// LS Electric XG5000 project: Maycatnhom_Q9
// PLC NewPLC

PROGRAM Orijine Git (task: Scan Program)

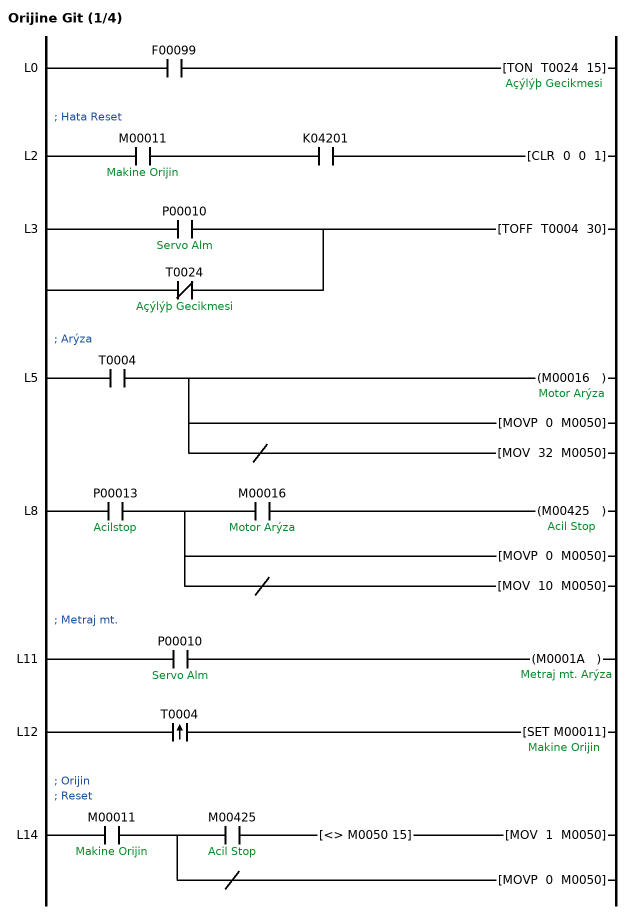
; L0
LOAD      F00099
TON       T0024 15	// Açýlýþ Gecikmesi
// Hata Reset
; L2
LOAD      M00011	// Makine Orijin
AND       K04201
CLR       0 0 1
; L3
LOAD      P00010	// Servo Alm
OR NOT    T0024	// Açýlýþ Gecikmesi
TOFF      T0004 30
; L5
LOAD      T0004
OUT       M00016	// Motor Arýza
MOVP      0 M0050
NOT
MOV       32 M0050
// output comment: Arýza
; L8
LOAD      P00013	// Acilstop
MPUSH
AND       M00016	// Motor Arýza
OUT       M00425	// Acil Stop
MPOP
MOVP      0 M0050
NOT
MOV       10 M0050
; L11
LOAD      P00010	// Servo Alm
OUT       M0001A	// Metraj mt. Arýza
// output comment: Metraj mt.
; L12
LOADP     T0004
SET       M00011	// Makine Orijin
// Orijin
; L14
LOAD      M00011	// Makine Orijin
MPUSH
AND       M00425	// Acil Stop
AND<>     M0050 15
MOV       1 M0050
MPOP
NOT
MOVP      0 M0050
// output comment: Reset

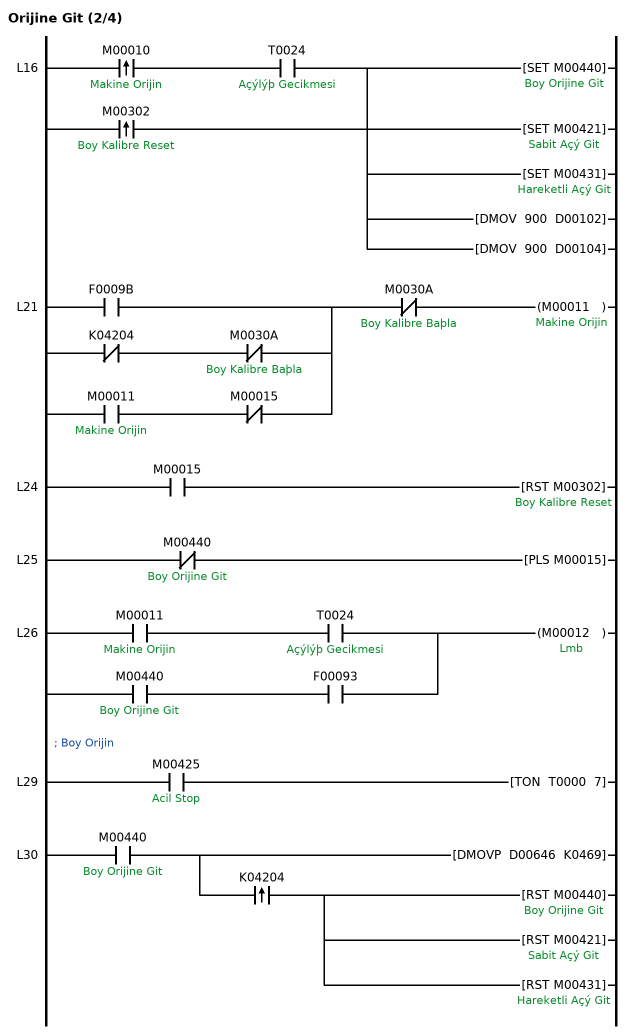
; L16
LOADP     M00010	// Makine Orijin
AND       T0024	// Açýlýþ Gecikmesi
ORP       M00302	// Boy Kalibre Reset
SET       M00440	// Boy Orijine Git
SET       M00421	// Sabit Açý Git
SET       M00431	// Hareketli Açý Git
DMOV      900 D00102
DMOV      900 D00104
; L21
LOAD      F0009B
LOAD NOT  K04204
AND NOT   M0030A	// Boy Kalibre Baþla
OR LOAD
LOAD      M00011	// Makine Orijin
AND NOT   M00015
OR LOAD
AND NOT   M0030A	// Boy Kalibre Baþla
OUT       M00011	// Makine Orijin
; L24
LOAD      M00015
RST       M00302	// Boy Kalibre Reset
; L25
LOAD NOT  M00440	// Boy Orijine Git
OUTP      M00015
; L26
LOAD      M00011	// Makine Orijin
AND       T0024	// Açýlýþ Gecikmesi
LOAD      M00440	// Boy Orijine Git
AND       F00093
OR LOAD
OUT       M00012	// Lmb
// Boy Orijin
; L29
LOAD      M00425	// Acil Stop
TON       T0000 7
; L30
LOAD      M00440	// Boy Orijine Git
DMOVP     D00646 K0469
ANDP      K04204
RST       M00440	// Boy Orijine Git
RST       M00421	// Sabit Açý Git
RST       M00431	// Hareketli Açý Git

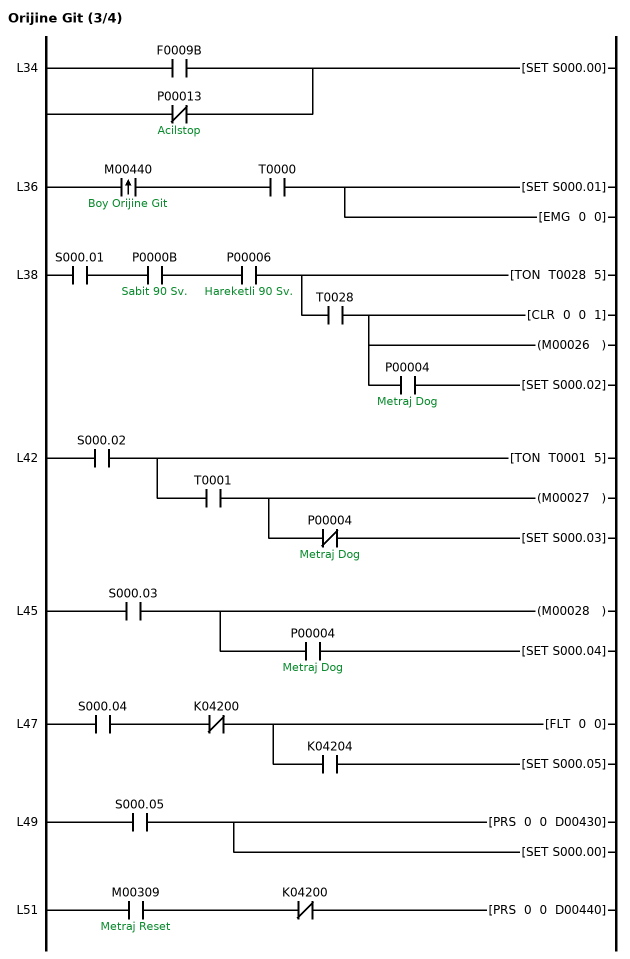
; L34
LOAD      F0009B
OR NOT    P00013	// Acilstop
SET       S000.00
; L36
LOADP     M00440	// Boy Orijine Git
AND       T0000
SET       S000.01
EMG       0 0
; L38
LOAD      S000.01
AND       P0000B	// Sabit 90 Sv.
AND       P00006	// Hareketli 90 Sv.
TON       T0028 5
AND       T0028
CLR       0 0 1
OUT       M00026
AND       P00004	// Metraj Dog
SET       S000.02
; L42
LOAD      S000.02
TON       T0001 5
AND       T0001
OUT       M00027
AND NOT   P00004	// Metraj Dog
SET       S000.03
; L45
LOAD      S000.03
OUT       M00028
AND       P00004	// Metraj Dog
SET       S000.04
; L47
LOAD      S000.04
AND NOT   K04200
FLT       0 0
AND       K04204
SET       S000.05
; L49
LOAD      S000.05
PRS       0 0 D00430
SET       S000.00
; L51
LOAD      M00309	// Metraj Reset
AND NOT   K04200
PRS       0 0 D00440

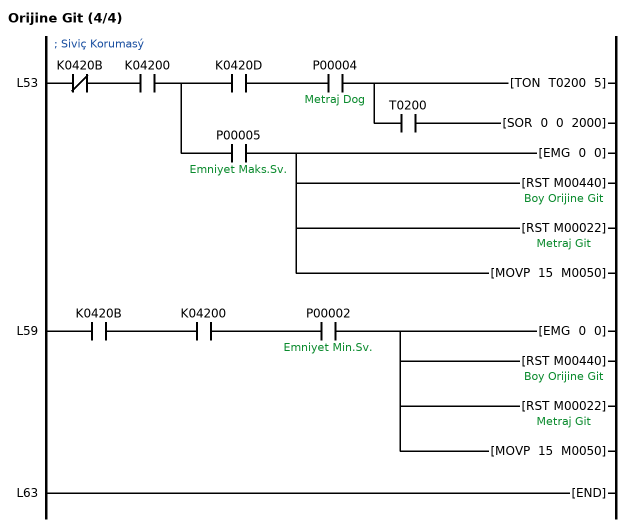
// Siviç Korumasý
; L53
LOAD NOT  K0420B
AND       K04200
MPUSH
AND       K0420D
AND       P00004	// Metraj Dog
TON       T0200 5
AND       T0200
SOR       0 0 2000
MPOP
AND       P00005	// Emniyet Maks.Sv.
EMG       0 0
RST       M00440	// Boy Orijine Git
RST       M00022	// Metraj Git
MOVP      15 M0050
; L59
LOAD      K0420B
AND       K04200
AND       P00002	// Emniyet Min.Sv.
EMG       0 0
RST       M00440	// Boy Orijine Git
RST       M00022	// Metraj Git
MOVP      15 M0050
; L63
END

PROGRAM Testere (task: Scan Program)

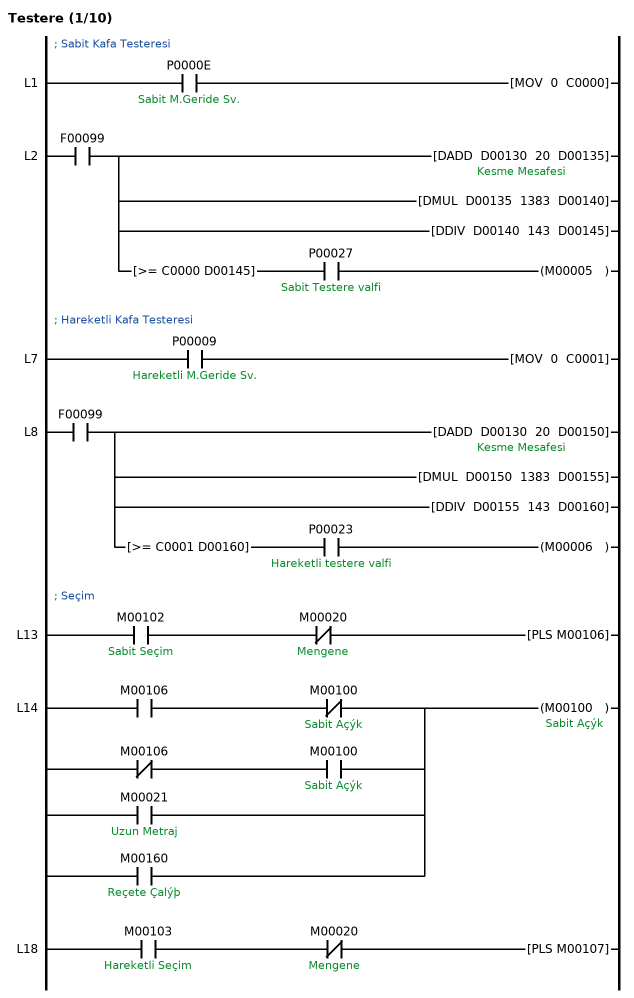
// Sabit Kafa Testeresi
; L1
LOAD      P0000E	// Sabit M.Geride Sv.
MOV       0 C0000
; L2
LOAD      F00099
DADD      D00130 20 D00135	// Kesme Mesafesi
DMUL      D00135 1383 D00140
DDIV      D00140 143 D00145
AND>=     C0000 D00145
AND       P00027	// Sabit Testere valfi
OUT       M00005
// Hareketli Kafa Testeresi
; L7
LOAD      P00009	// Hareketli M.Geride Sv.
MOV       0 C0001
; L8
LOAD      F00099
DADD      D00130 20 D00150	// Kesme Mesafesi
DMUL      D00150 1383 D00155
DDIV      D00155 143 D00160
AND>=     C0001 D00160
AND       P00023	// Hareketli testere valfi
OUT       M00006
// Seçim
; L13
LOAD      M00102	// Sabit Seçim
AND NOT   M00020	// Mengene
OUTP      M00106
; L14
LOAD      M00106
AND NOT   M00100	// Sabit Açýk
LOAD NOT  M00106
AND       M00100	// Sabit Açýk
OR LOAD
OR        M00021	// Uzun Metraj
OR        M00160	// Reçete Çalýþ
OUT       M00100	// Sabit Açýk
; L18
LOAD      M00103	// Hareketli Seçim
AND NOT   M00020	// Mengene
OUTP      M00107

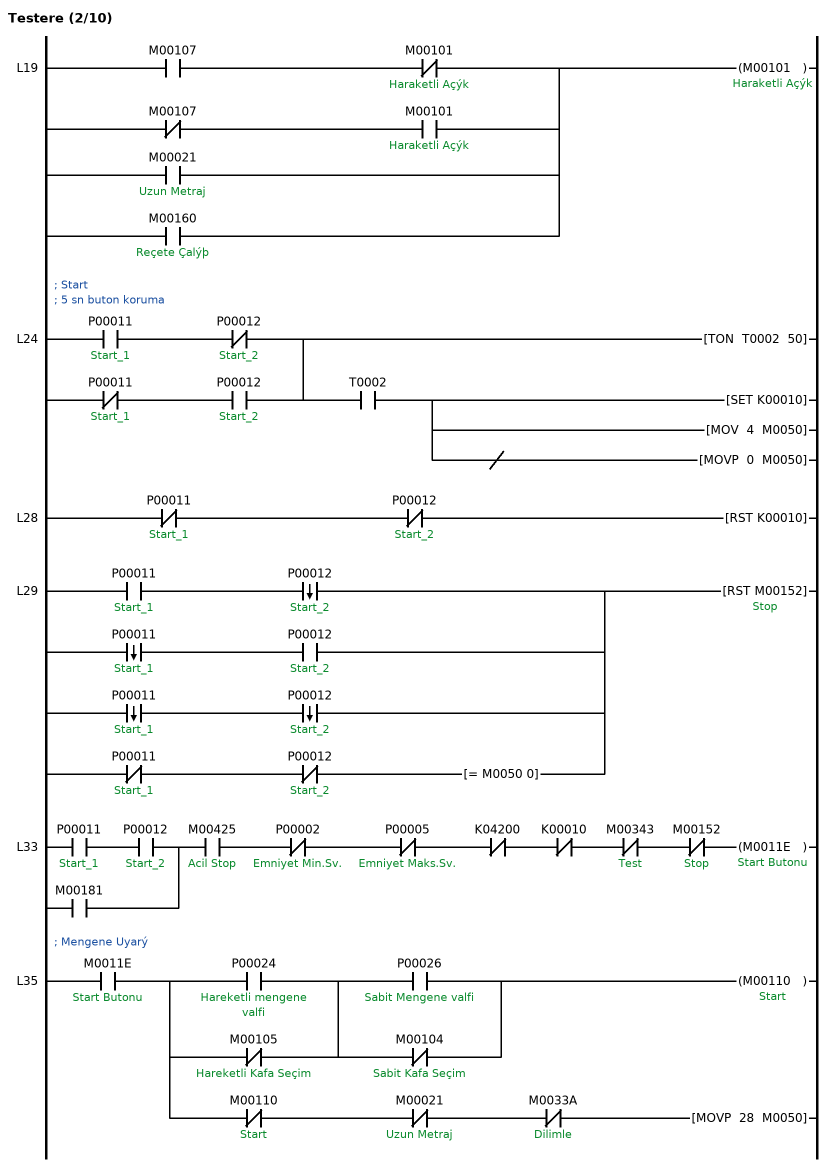
; L19
LOAD      M00107
AND NOT   M00101	// Haraketli Açýk
LOAD NOT  M00107
AND       M00101	// Haraketli Açýk
OR LOAD
OR        M00021	// Uzun Metraj
OR        M00160	// Reçete Çalýþ
OUT       M00101	// Haraketli Açýk
// Start
; L24
LOAD      P00011	// Start_1
AND NOT   P00012	// Start_2
LOAD NOT  P00011	// Start_1
AND       P00012	// Start_2
OR LOAD
TON       T0002 50
AND       T0002
SET       K00010
MOV       4 M0050
NOT
MOVP      0 M0050
// output comment: 5 sn buton koruma
; L28
LOAD NOT  P00011	// Start_1
AND NOT   P00012	// Start_2
RST       K00010
; L29
LOAD      P00011	// Start_1
ANDN      P00012	// Start_2
LOADN     P00011	// Start_1
AND       P00012	// Start_2
OR LOAD
LOADN     P00011	// Start_1
ANDN      P00012	// Start_2
OR LOAD
LOAD NOT  P00011	// Start_1
AND NOT   P00012	// Start_2
AND=      M0050 0
OR LOAD
RST       M00152	// Stop
; L33
LOAD      P00011	// Start_1
AND       P00012	// Start_2
OR        M00181
AND       M00425	// Acil Stop
AND NOT   P00002	// Emniyet Min.Sv.
AND NOT   P00005	// Emniyet Maks.Sv.
AND NOT   K04200
AND NOT   K00010
AND NOT   M00343	// Test
AND NOT   M00152	// Stop
OUT       M0011E	// Start Butonu
; L35
LOAD      M0011E	// Start Butonu
MPUSH
LOAD      P00024	// Hareketli mengene valfi
OR NOT    M00105	// Hareketli Kafa Seçim
AND LOAD
LOAD      P00026	// Sabit Mengene valfi
OR NOT    M00104	// Sabit Kafa Seçim
AND LOAD
OUT       M00110	// Start
MPOP
AND NOT   M00110	// Start
AND NOT   M00021	// Uzun Metraj
AND NOT   M0033A	// Dilimle
MOVP      28 M0050
// output comment: Mengene Uyarý

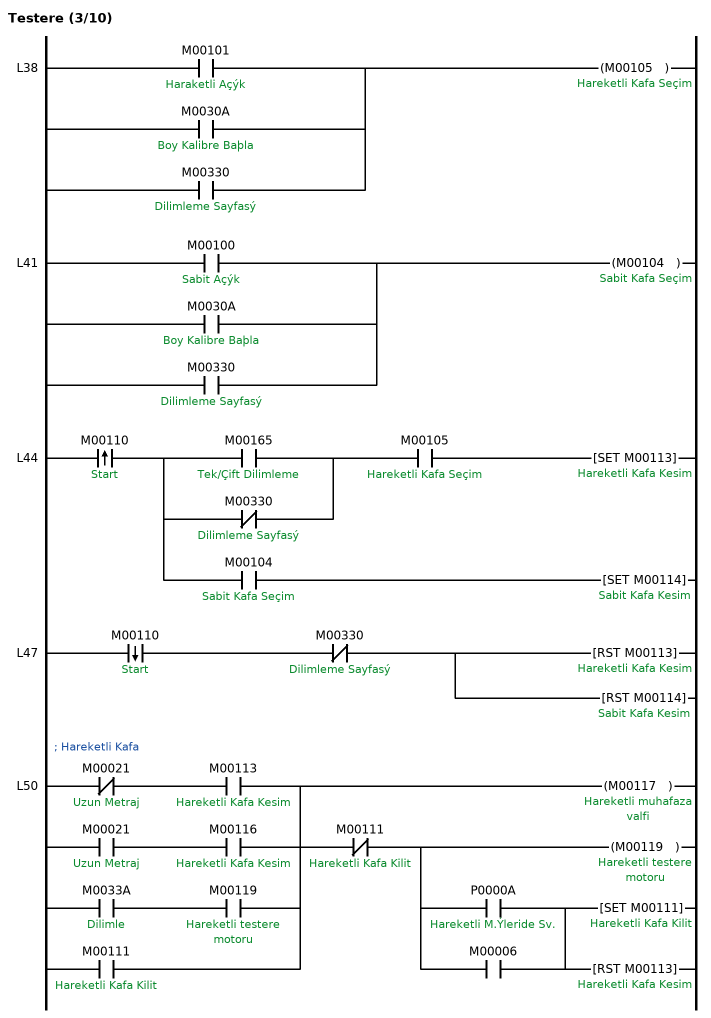
; L38
LOAD      M00101	// Haraketli Açýk
OR        M0030A	// Boy Kalibre Baþla
OR        M00330	// Dilimleme Sayfasý
OUT       M00105	// Hareketli Kafa Seçim
; L41
LOAD      M00100	// Sabit Açýk
OR        M0030A	// Boy Kalibre Baþla
OR        M00330	// Dilimleme Sayfasý
OUT       M00104	// Sabit Kafa Seçim
; L44
LOADP     M00110	// Start
MPUSH
LOAD      M00165	// Tek/Çift Dilimleme
OR NOT    M00330	// Dilimleme Sayfasý
AND LOAD
AND       M00105	// Hareketli Kafa Seçim
SET       M00113	// Hareketli Kafa Kesim
MPOP
AND       M00104	// Sabit Kafa Seçim
SET       M00114	// Sabit Kafa Kesim
; L47
LOADN     M00110	// Start
AND NOT   M00330	// Dilimleme Sayfasý
RST       M00113	// Hareketli Kafa Kesim
RST       M00114	// Sabit Kafa Kesim
// Hareketli Kafa
; L50
LOAD NOT  M00021	// Uzun Metraj
AND       M00113	// Hareketli Kafa Kesim
LOAD      M00021	// Uzun Metraj
AND       M00116	// Hareketli Kafa Kesim
OR LOAD
LOAD      M0033A	// Dilimle
AND       M00119	// Hareketli testere motoru
OR LOAD
OR        M00111	// Hareketli Kafa Kilit
OUT       M00117	// Hareketli muhafaza valfi
AND NOT   M00111	// Hareketli Kafa Kilit
OUT       M00119	// Hareketli testere motoru
LOAD      P0000A	// Hareketli M.Ýleride Sv.
OR        M00006
AND LOAD
SET       M00111	// Hareketli Kafa Kilit
RST       M00113	// Hareketli Kafa Kesim

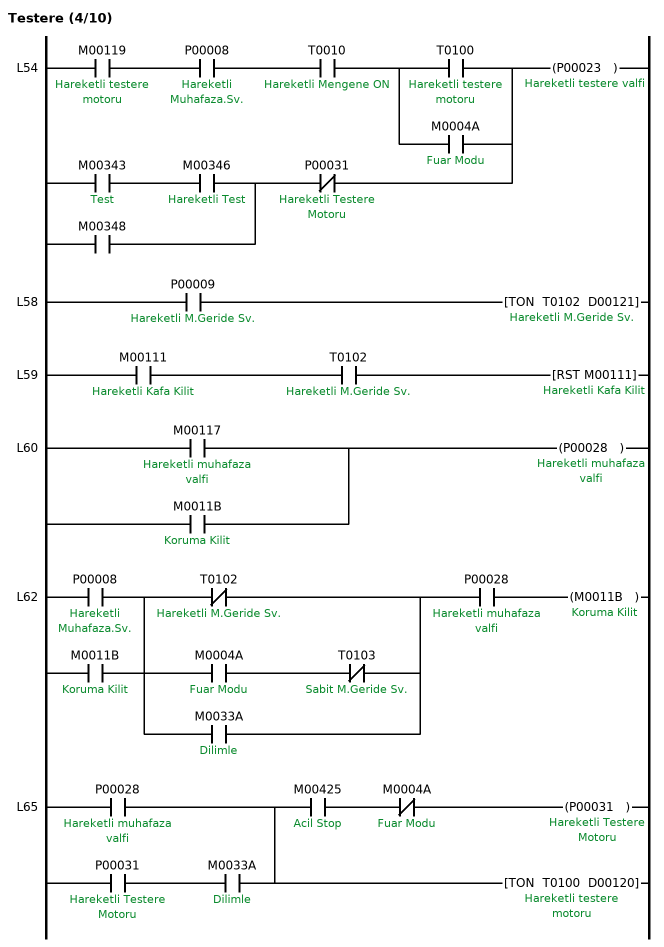
; L54
LOAD      M00119	// Hareketli testere motoru
AND       P00008	// Hareketli Muhafaza.Sv.
AND       T0010	// Hareketli Mengene ON
LOAD      T0100	// Hareketli testere motoru
OR        M0004A	// Fuar Modu
AND LOAD
LOAD      M00343	// Test
AND       M00346	// Hareketli Test
OR        M00348
AND NOT   P00031	// Hareketli Testere Motoru
OR LOAD
OUT       P00023	// Hareketli testere valfi
; L58
LOAD      P00009	// Hareketli M.Geride Sv.
TON       T0102 D00121	// Hareketli M.Geride Sv.
; L59
LOAD      M00111	// Hareketli Kafa Kilit
AND       T0102	// Hareketli M.Geride Sv.
RST       M00111	// Hareketli Kafa Kilit
; L60
LOAD      M00117	// Hareketli muhafaza valfi
OR        M0011B	// Koruma Kilit
OUT       P00028	// Hareketli muhafaza valfi
; L62
LOAD      P00008	// Hareketli Muhafaza.Sv.
OR        M0011B	// Koruma Kilit
LOAD NOT  T0102	// Hareketli M.Geride Sv.
LOAD      M0004A	// Fuar Modu
AND NOT   T0103	// Sabit M.Geride Sv.
OR LOAD
OR        M0033A	// Dilimle
AND LOAD
AND       P00028	// Hareketli muhafaza valfi
OUT       M0011B	// Koruma Kilit
; L65
LOAD      P00028	// Hareketli muhafaza valfi
LOAD      P00031	// Hareketli Testere Motoru
AND       M0033A	// Dilimle
OR LOAD
MPUSH
AND       M00425	// Acil Stop
AND NOT   M0004A	// Fuar Modu
OUT       P00031	// Hareketli Testere Motoru
MPOP
TON       T0100 D00120	// Hareketli testere motoru

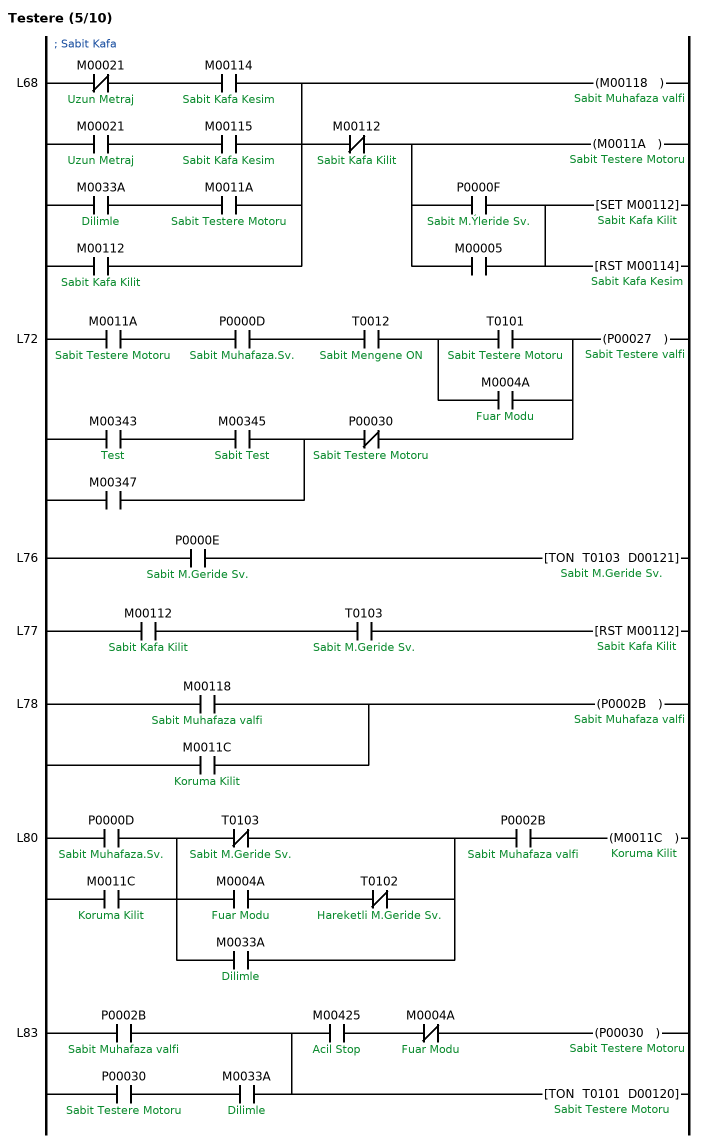
// Sabit Kafa
; L68
LOAD NOT  M00021	// Uzun Metraj
AND       M00114	// Sabit Kafa Kesim
LOAD      M00021	// Uzun Metraj
AND       M00115	// Sabit Kafa Kesim
OR LOAD
LOAD      M0033A	// Dilimle
AND       M0011A	// Sabit Testere Motoru
OR LOAD
OR        M00112	// Sabit Kafa Kilit
OUT       M00118	// Sabit Muhafaza valfi
AND NOT   M00112	// Sabit Kafa Kilit
OUT       M0011A	// Sabit Testere Motoru
LOAD      P0000F	// Sabit M.Ýleride Sv.
OR        M00005
AND LOAD
SET       M00112	// Sabit Kafa Kilit
RST       M00114	// Sabit Kafa Kesim
; L72
LOAD      M0011A	// Sabit Testere Motoru
AND       P0000D	// Sabit Muhafaza.Sv.
AND       T0012	// Sabit Mengene ON
LOAD      T0101	// Sabit Testere Motoru
OR        M0004A	// Fuar Modu
AND LOAD
LOAD      M00343	// Test
AND       M00345	// Sabit Test
OR        M00347
AND NOT   P00030	// Sabit Testere Motoru
OR LOAD
OUT       P00027	// Sabit Testere valfi
; L76
LOAD      P0000E	// Sabit M.Geride Sv.
TON       T0103 D00121	// Sabit M.Geride Sv.
; L77
LOAD      M00112	// Sabit Kafa Kilit
AND       T0103	// Sabit M.Geride Sv.
RST       M00112	// Sabit Kafa Kilit
; L78
LOAD      M00118	// Sabit Muhafaza valfi
OR        M0011C	// Koruma Kilit
OUT       P0002B	// Sabit Muhafaza valfi
; L80
LOAD      P0000D	// Sabit Muhafaza.Sv.
OR        M0011C	// Koruma Kilit
LOAD NOT  T0103	// Sabit M.Geride Sv.
LOAD      M0004A	// Fuar Modu
AND NOT   T0102	// Hareketli M.Geride Sv.
OR LOAD
OR        M0033A	// Dilimle
AND LOAD
AND       P0002B	// Sabit Muhafaza valfi
OUT       M0011C	// Koruma Kilit
; L83
LOAD      P0002B	// Sabit Muhafaza valfi
LOAD      P00030	// Sabit Testere Motoru
AND       M0033A	// Dilimle
OR LOAD
MPUSH
AND       M00425	// Acil Stop
AND NOT   M0004A	// Fuar Modu
OUT       P00030	// Sabit Testere Motoru
MPOP
TON       T0101 D00120	// Sabit Testere Motoru

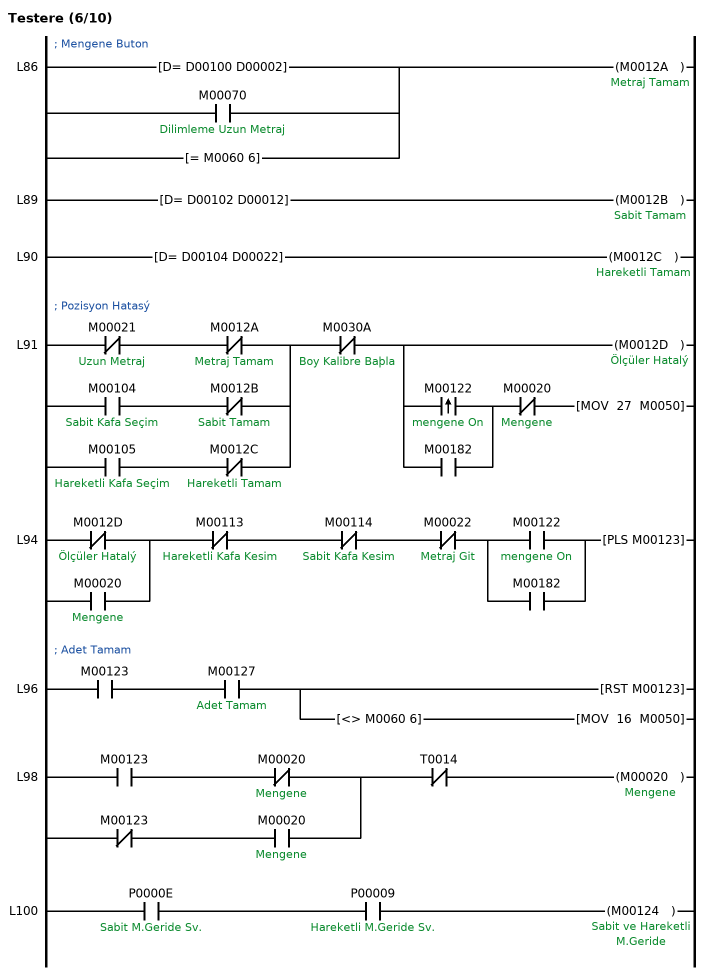
// Mengene Buton
; L86
LOADD=    D00100 D00002
OR        M00070	// Dilimleme Uzun Metraj
OR=       M0060 6
OUT       M0012A	// Metraj Tamam
; L89
LOADD=    D00102 D00012
OUT       M0012B	// Sabit Tamam
; L90
LOADD=    D00104 D00022
OUT       M0012C	// Hareketli Tamam
; L91
LOAD NOT  M00021	// Uzun Metraj
AND NOT   M0012A	// Metraj Tamam
LOAD      M00104	// Sabit Kafa Seçim
AND NOT   M0012B	// Sabit Tamam
OR LOAD
LOAD      M00105	// Hareketli Kafa Seçim
AND NOT   M0012C	// Hareketli Tamam
OR LOAD
AND NOT   M0030A	// Boy Kalibre Baþla
OUT       M0012D	// Ölçüler Hatalý
LOADP     M00122	// mengene On
OR        M00182
AND LOAD
AND NOT   M00020	// Mengene
MOV       27 M0050
// output comment: Pozisyon Hatasý
; L94
LOAD NOT  M0012D	// Ölçüler Hatalý
OR        M00020	// Mengene
AND NOT   M00113	// Hareketli Kafa Kesim
AND NOT   M00114	// Sabit Kafa Kesim
AND NOT   M00022	// Metraj Git
LOAD      M00122	// mengene On
OR        M00182
AND LOAD
OUTP      M00123
; L96
LOAD      M00123
AND       M00127	// Adet Tamam
RST       M00123
AND<>     M0060 6
MOV       16 M0050
// output comment: Adet Tamam
; L98
LOAD      M00123
AND NOT   M00020	// Mengene
LOAD NOT  M00123
AND       M00020	// Mengene
OR LOAD
AND NOT   T0014
OUT       M00020	// Mengene
; L100
LOAD      P0000E	// Sabit M.Geride Sv.
AND       P00009	// Hareketli M.Geride Sv.
OUT       M00124	// Sabit ve Hareketli M.Geride

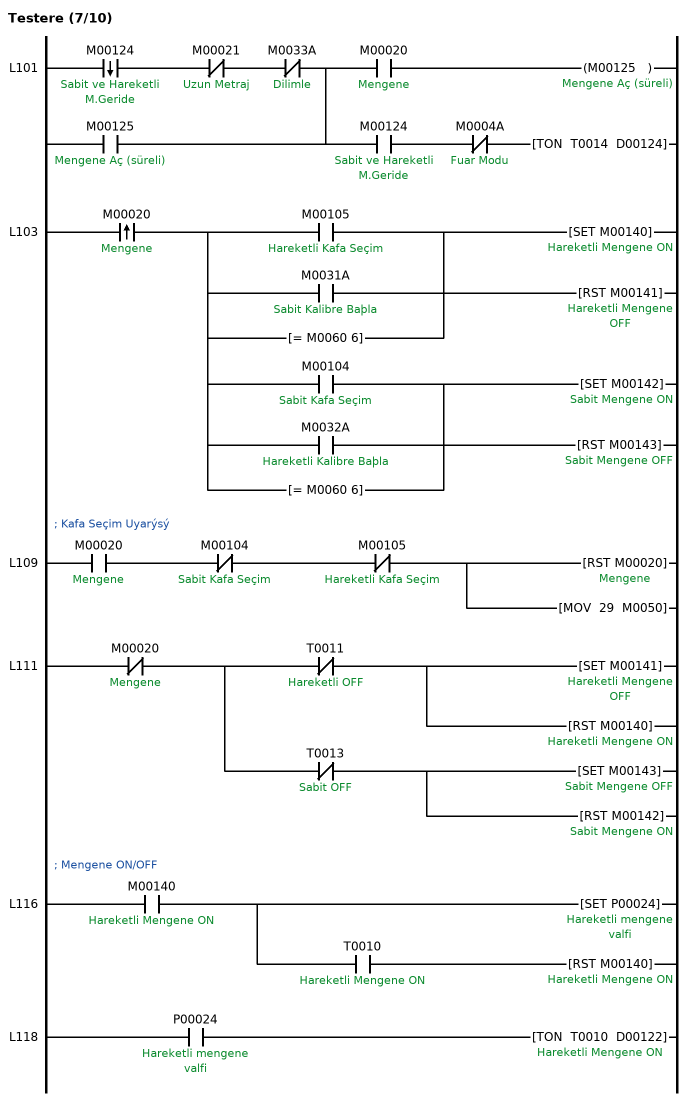
; L101
LOADN     M00124	// Sabit ve Hareketli M.Geride
AND NOT   M00021	// Uzun Metraj
AND NOT   M0033A	// Dilimle
OR        M00125	// Mengene Aç (süreli)
MPUSH
AND       M00020	// Mengene
OUT       M00125	// Mengene Aç (süreli)
MPOP
AND       M00124	// Sabit ve Hareketli M.Geride
AND NOT   M0004A	// Fuar Modu
TON       T0014 D00124
; L103
LOADP     M00020	// Mengene
MPUSH
LOAD      M00105	// Hareketli Kafa Seçim
OR        M0031A	// Sabit Kalibre Baþla
OR=       M0060 6
AND LOAD
SET       M00140	// Hareketli Mengene ON
RST       M00141	// Hareketli Mengene OFF
MPOP
LOAD      M00104	// Sabit Kafa Seçim
OR        M0032A	// Hareketli Kalibre Baþla
OR=       M0060 6
AND LOAD
SET       M00142	// Sabit Mengene ON
RST       M00143	// Sabit Mengene OFF
; L109
LOAD      M00020	// Mengene
AND NOT   M00104	// Sabit Kafa Seçim
AND NOT   M00105	// Hareketli Kafa Seçim
RST       M00020	// Mengene
MOV       29 M0050
// output comment: Kafa Seçim Uyarýsý
; L111
LOAD NOT  M00020	// Mengene
MPUSH
AND NOT   T0011	// Hareketli OFF
SET       M00141	// Hareketli Mengene OFF
RST       M00140	// Hareketli Mengene ON
MPOP
AND NOT   T0013	// Sabit OFF
SET       M00143	// Sabit Mengene OFF
RST       M00142	// Sabit Mengene ON
// Mengene ON/OFF
; L116
LOAD      M00140	// Hareketli Mengene ON
SET       P00024	// Hareketli mengene valfi
AND       T0010	// Hareketli Mengene ON
RST       M00140	// Hareketli Mengene ON
; L118
LOAD      P00024	// Hareketli mengene valfi
TON       T0010 D00122	// Hareketli Mengene ON

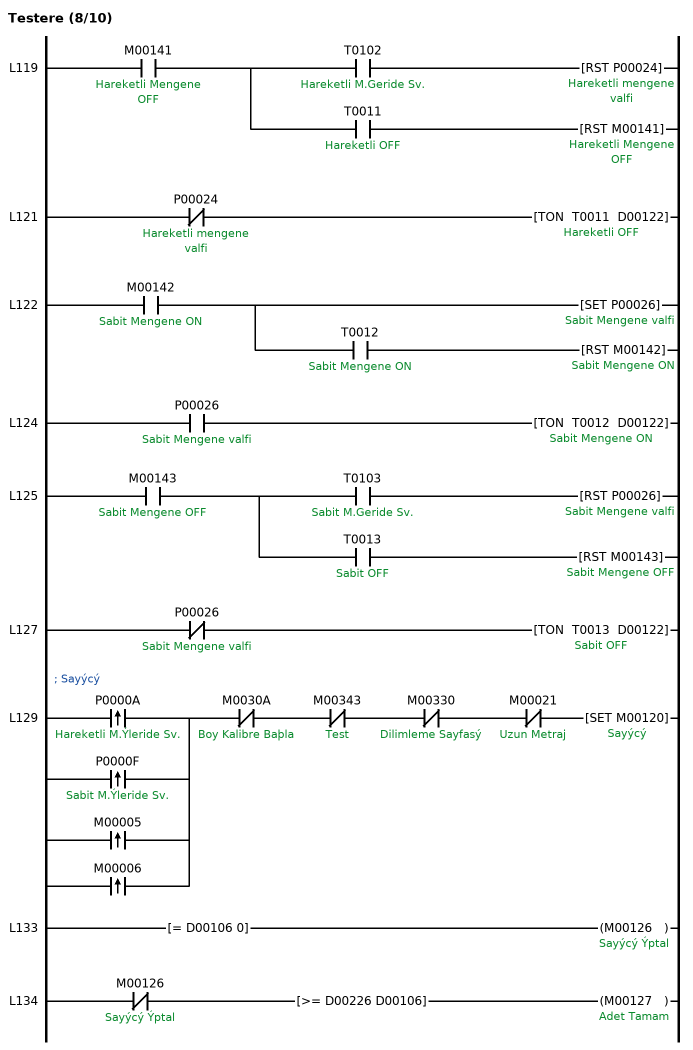
; L119
LOAD      M00141	// Hareketli Mengene OFF
MPUSH
AND       T0102	// Hareketli M.Geride Sv.
RST       P00024	// Hareketli mengene valfi
MPOP
AND       T0011	// Hareketli OFF
RST       M00141	// Hareketli Mengene OFF
; L121
LOAD NOT  P00024	// Hareketli mengene valfi
TON       T0011 D00122	// Hareketli OFF
; L122
LOAD      M00142	// Sabit Mengene ON
SET       P00026	// Sabit Mengene valfi
AND       T0012	// Sabit Mengene ON
RST       M00142	// Sabit Mengene ON
; L124
LOAD      P00026	// Sabit Mengene valfi
TON       T0012 D00122	// Sabit Mengene ON
; L125
LOAD      M00143	// Sabit Mengene OFF
MPUSH
AND       T0103	// Sabit M.Geride Sv.
RST       P00026	// Sabit Mengene valfi
MPOP
AND       T0013	// Sabit OFF
RST       M00143	// Sabit Mengene OFF
; L127
LOAD NOT  P00026	// Sabit Mengene valfi
TON       T0013 D00122	// Sabit OFF
// Sayýcý
; L129
LOADP     P0000A	// Hareketli M.Ýleride Sv.
ORP       P0000F	// Sabit M.Ýleride Sv.
ORP       M00005
ORP       M00006
AND NOT   M0030A	// Boy Kalibre Baþla
AND NOT   M00343	// Test
AND NOT   M00330	// Dilimleme Sayfasý
AND NOT   M00021	// Uzun Metraj
SET       M00120	// Sayýcý
; L133
LOAD=     D00106 0
OUT       M00126	// Sayýcý Ýptal
; L134
LOAD NOT  M00126	// Sayýcý Ýptal
AND>=     D00226 D00106
OUT       M00127	// Adet Tamam

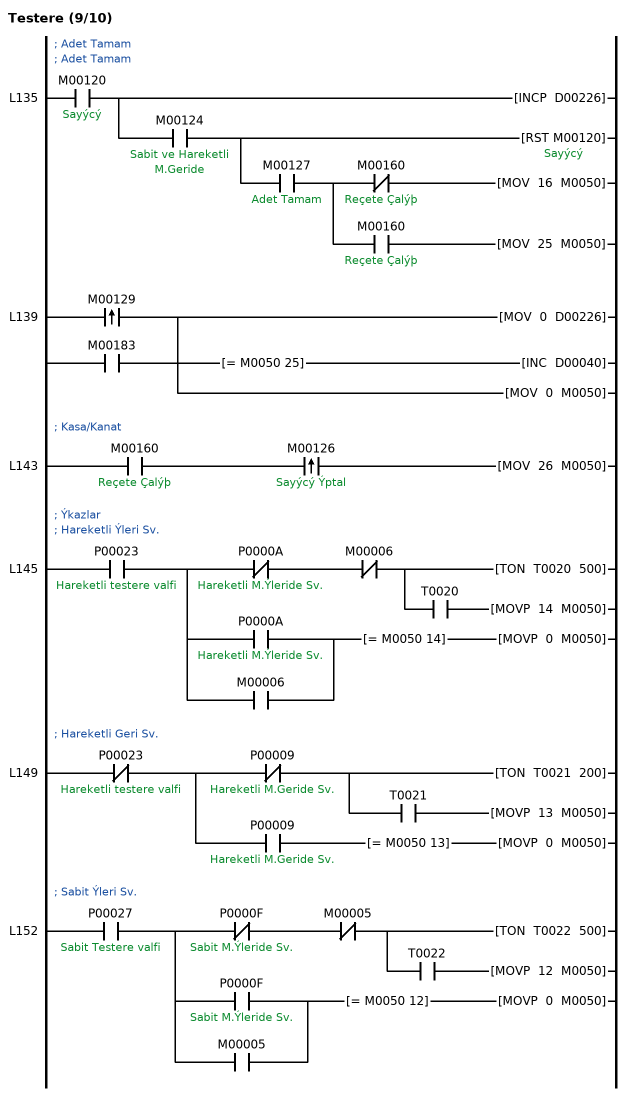
; L135
LOAD      M00120	// Sayýcý
INCP      D00226
AND       M00124	// Sabit ve Hareketli M.Geride
RST       M00120	// Sayýcý
AND       M00127	// Adet Tamam
MPUSH
AND NOT   M00160	// Reçete Çalýþ
MOV       16 M0050
MPOP
AND       M00160	// Reçete Çalýþ
MOV       25 M0050
// output comment: Adet Tamam
// output comment: Adet Tamam
; L139
LOADP     M00129
OR        M00183
MOV       0 D00226
MPUSH
AND=      M0050 25
INC       D00040
MPOP
MOV       0 M0050
// Kasa/Kanat
; L143
LOAD      M00160	// Reçete Çalýþ
ANDP      M00126	// Sayýcý Ýptal
MOV       26 M0050
// Ýkazlar
; L145
LOAD      P00023	// Hareketli testere valfi
MPUSH
AND NOT   P0000A	// Hareketli M.Ýleride Sv.
AND NOT   M00006
TON       T0020 500
AND       T0020
MOVP      14 M0050
MPOP
LOAD      P0000A	// Hareketli M.Ýleride Sv.
OR        M00006
AND LOAD
AND=      M0050 14
MOVP      0 M0050
// output comment: Hareketli Ýleri Sv.
; L149
LOAD NOT  P00023	// Hareketli testere valfi
MPUSH
AND NOT   P00009	// Hareketli M.Geride Sv.
TON       T0021 200
AND       T0021
MOVP      13 M0050
MPOP
AND       P00009	// Hareketli M.Geride Sv.
AND=      M0050 13
MOVP      0 M0050
// output comment: Hareketli Geri Sv.
; L152
LOAD      P00027	// Sabit Testere valfi
MPUSH
AND NOT   P0000F	// Sabit M.Ýleride Sv.
AND NOT   M00005
TON       T0022 500
AND       T0022
MOVP      12 M0050
MPOP
LOAD      P0000F	// Sabit M.Ýleride Sv.
OR        M00005
AND LOAD
AND=      M0050 12
MOVP      0 M0050
// output comment: Sabit Ýleri Sv.

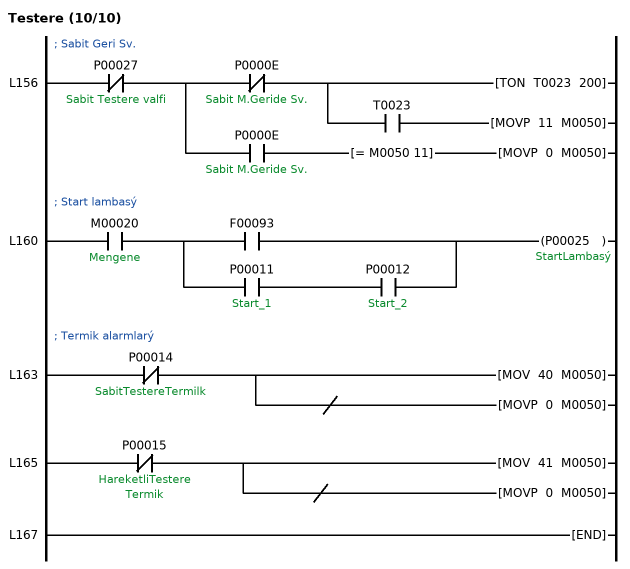
; L156
LOAD NOT  P00027	// Sabit Testere valfi
MPUSH
AND NOT   P0000E	// Sabit M.Geride Sv.
TON       T0023 200
AND       T0023
MOVP      11 M0050
MPOP
AND       P0000E	// Sabit M.Geride Sv.
AND=      M0050 11
MOVP      0 M0050
// output comment: Sabit Geri Sv.
// Start lambasý
; L160
LOAD      M00020	// Mengene
LOAD      F00093
LOAD      P00011	// Start_1
AND       P00012	// Start_2
OR LOAD
AND LOAD
OUT       P00025	// StartLambasý
// Termik alarmlarý
; L163
LOAD NOT  P00014	// SabitTestereTermilk
MOV       40 M0050
NOT
MOVP      0 M0050
; L165
LOAD NOT  P00015	// HareketliTestereTermik
MOV       41 M0050
NOT
MOVP      0 M0050
; L167
END

PROGRAM Metraj Kalibrasyonu (task: Scan Program)

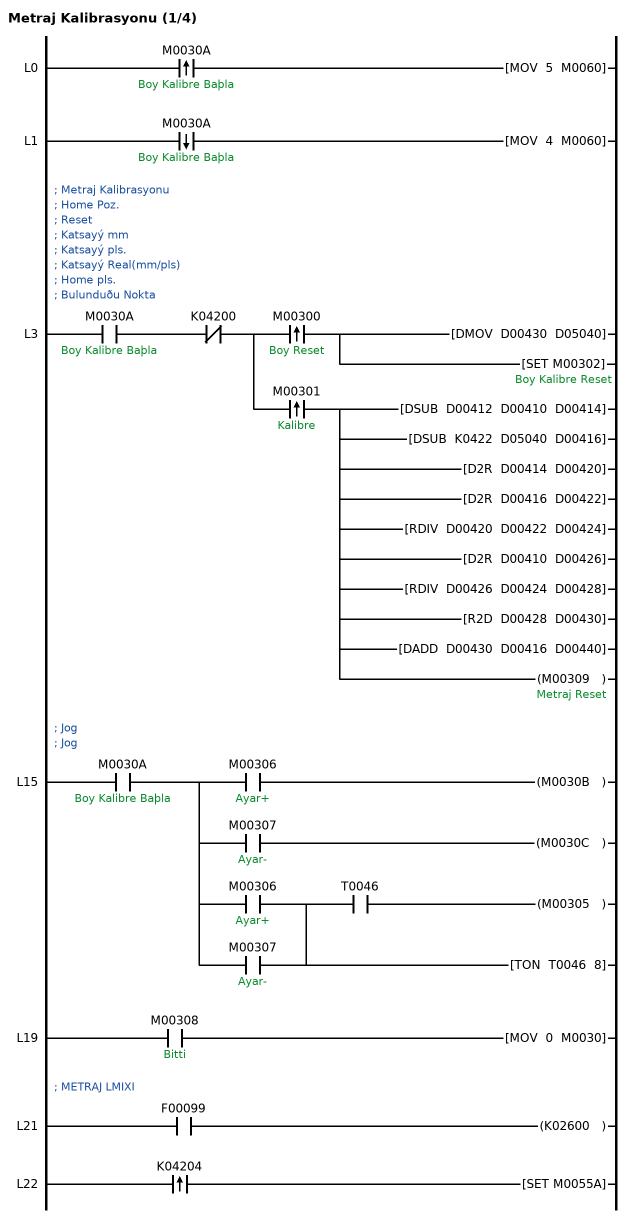
; L0
LOADP     M0030A	// Boy Kalibre Baþla
MOV       5 M0060
; L1
LOADN     M0030A	// Boy Kalibre Baþla
MOV       4 M0060
// Metraj Kalibrasyonu
; L3
LOAD      M0030A	// Boy Kalibre Baþla
AND NOT   K04200
MPUSH
ANDP      M00300	// Boy Reset
DMOV      D00430 D05040
SET       M00302	// Boy Kalibre Reset
MPOP
ANDP      M00301	// Kalibre
DSUB      D00412 D00410 D00414
DSUB      K0422 D05040 D00416
D2R       D00414 D00420
D2R       D00416 D00422
RDIV      D00420 D00422 D00424
D2R       D00410 D00426
RDIV      D00426 D00424 D00428
R2D       D00428 D00430
DADD      D00430 D00416 D00440
OUT       M00309	// Metraj Reset
// output comment: Home Poz.
// output comment: Reset
// output comment: Katsayý mm
// output comment: Katsayý pls.
// output comment: Katsayý Real(mm/pls)
// output comment: Home pls.
// output comment: Bulunduðu Nokta
; L15
LOAD      M0030A	// Boy Kalibre Baþla
MPUSH
AND       M00306	// Ayar+
OUT       M0030B
MLOAD
AND       M00307	// Ayar-
OUT       M0030C
MPOP
LOAD      M00306	// Ayar+
OR        M00307	// Ayar-
AND LOAD
MPUSH
AND       T0046
OUT       M00305
MPOP
TON       T0046 8
// output comment: Jog
// output comment: Jog
; L19
LOAD      M00308	// Bitti
MOV       0 M0030
// METRAJ LMIXI
; L21
LOAD      F00099
OUT       K02600
; L22
LOADP     K04204
SET       M0055A

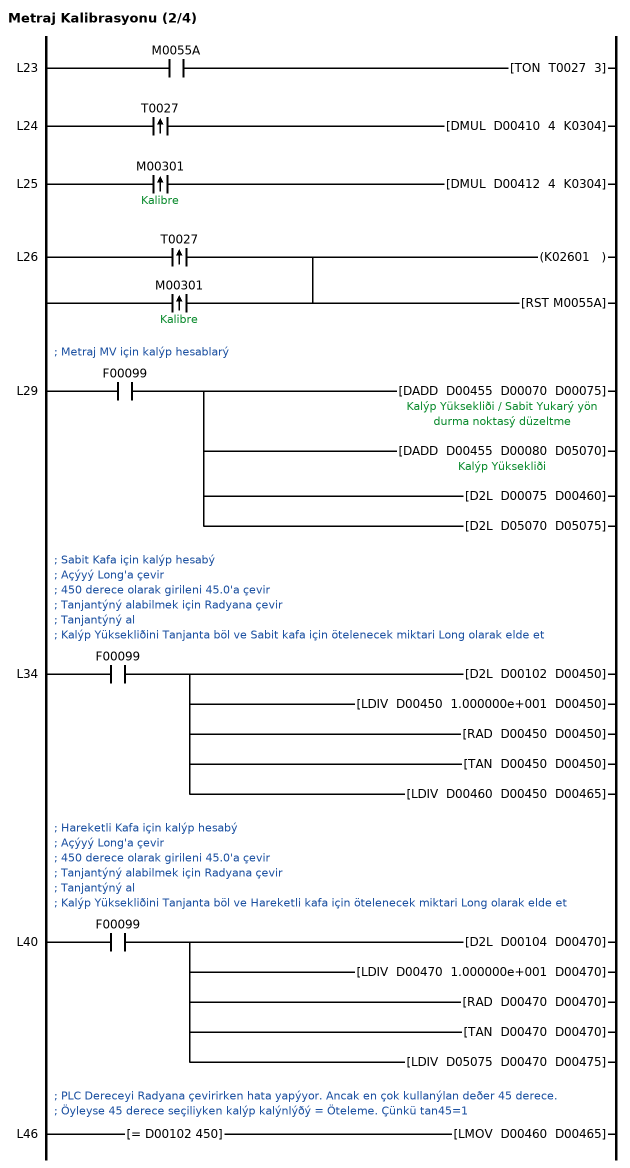
; L23
LOAD      M0055A
TON       T0027 3
; L24
LOADP     T0027
DMUL      D00410 4 K0304
; L25
LOADP     M00301	// Kalibre
DMUL      D00412 4 K0304
; L26
LOADP     T0027
ORP       M00301	// Kalibre
OUT       K02601
RST       M0055A
// Metraj MV için kalýp hesablarý
; L29
LOAD      F00099
DADD      D00455 D00070 D00075	// Kalýp Yüksekliði / Sabit Yukarý yön durma noktasý düzeltme
DADD      D00455 D00080 D05070	// Kalýp Yüksekliði
D2L       D00075 D00460
D2L       D05070 D05075
// Sabit Kafa için kalýp hesabý
; L34
LOAD      F00099
D2L       D00102 D00450
LDIV      D00450 1.000000e+001 D00450
RAD       D00450 D00450
TAN       D00450 D00450
LDIV      D00460 D00450 D00465
// output comment: Açýyý Long'a çevir
// output comment: 450 derece olarak girileni 45.0'a çevir
// output comment: Tanjantýný alabilmek için Radyana çevir
// output comment: Tanjantýný al
// output comment: Kalýp Yüksekliðini Tanjanta böl ve Sabit kafa için ötelenecek miktari Long olarak elde et
// Hareketli Kafa için kalýp hesabý
; L40
LOAD      F00099
D2L       D00104 D00470
LDIV      D00470 1.000000e+001 D00470
RAD       D00470 D00470
TAN       D00470 D00470
LDIV      D05075 D00470 D00475
// output comment: Açýyý Long'a çevir
// output comment: 450 derece olarak girileni 45.0'a çevir
// output comment: Tanjantýný alabilmek için Radyana çevir
// output comment: Tanjantýný al
// output comment: Kalýp Yüksekliðini Tanjanta böl ve Hareketli kafa için ötelenecek miktari Long olarak elde et
// PLC Dereceyi Radyana çevirirken hata yapýyor. Ancak en çok kullanýlan deðer 45 derece. Öyleyse 45 derece seçiliyken kalýp kalýnlýðý = Öteleme. Çünkü tan45=1
; L46
LOAD=     D00102 450
LMOV      D00460 D00465

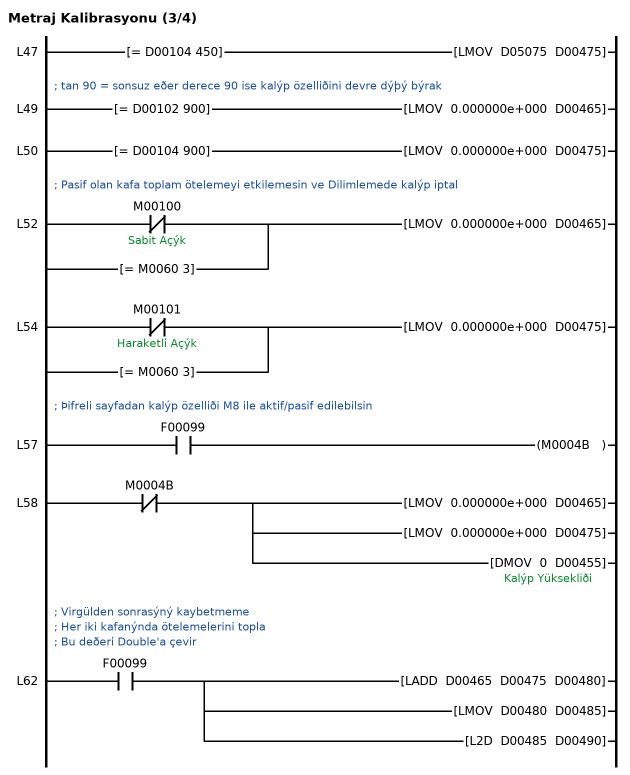
; L47
LOAD=     D00104 450
LMOV      D05075 D00475
// tan 90 = sonsuz eðer derece 90 ise kalýp özelliðini devre dýþý býrak
; L49
LOAD=     D00102 900
LMOV      0.000000e+000 D00465
; L50
LOAD=     D00104 900
LMOV      0.000000e+000 D00475
// Pasif olan kafa toplam ötelemeyi etkilemesin ve Dilimlemede kalýp iptal
; L52
LOAD NOT  M00100	// Sabit Açýk
OR=       M0060 3
LMOV      0.000000e+000 D00465
; L54
LOAD NOT  M00101	// Haraketli Açýk
OR=       M0060 3
LMOV      0.000000e+000 D00475
// Þifreli sayfadan kalýp özelliði M8 ile aktif/pasif edilebilsin
; L57
LOAD      F00099
OUT       M0004B
; L58
LOAD NOT  M0004B
LMOV      0.000000e+000 D00465
LMOV      0.000000e+000 D00475
DMOV      0 D00455	// Kalýp Yüksekliði
// Virgülden sonrasýný kaybetmeme
; L62
LOAD      F00099
LADD      D00465 D00475 D00480
LMOV      D00480 D00485
L2D       D00485 D00490
// output comment: Her iki kafanýnda ötelemelerini topla
// output comment: 
// output comment: Bu deðeri Double'a çevir

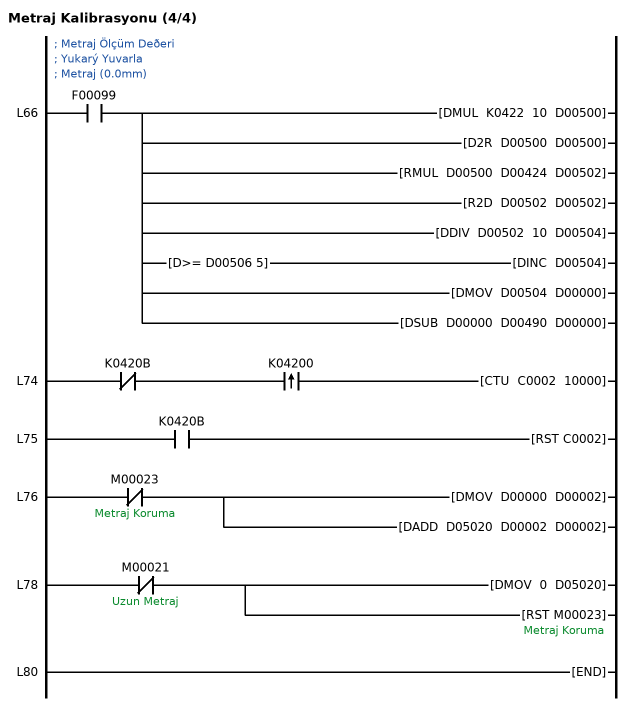
// Metraj Ölçüm Deðeri
; L66
LOAD      F00099
DMUL      K0422 10 D00500
D2R       D00500 D00500
RMUL      D00500 D00424 D00502
R2D       D00502 D00502
DDIV      D00502 10 D00504
MPUSH
ANDD>=    D00506 5
DINC      D00504
MPOP
DMOV      D00504 D00000
DSUB      D00000 D00490 D00000
// output comment: Yukarý Yuvarla
// output comment: Metraj (0.0mm)
; L74
LOAD NOT  K0420B
ANDP      K04200
CTU       C0002 10000
; L75
LOAD      K0420B
RST       C0002
; L76
LOAD NOT  M00023	// Metraj Koruma
DMOV      D00000 D00002
DADD      D05020 D00002 D00002
; L78
LOAD NOT  M00021	// Uzun Metraj
DMOV      0 D05020
RST       M00023	// Metraj Koruma
; L80
END

PROGRAM Git (task: Scan Program)

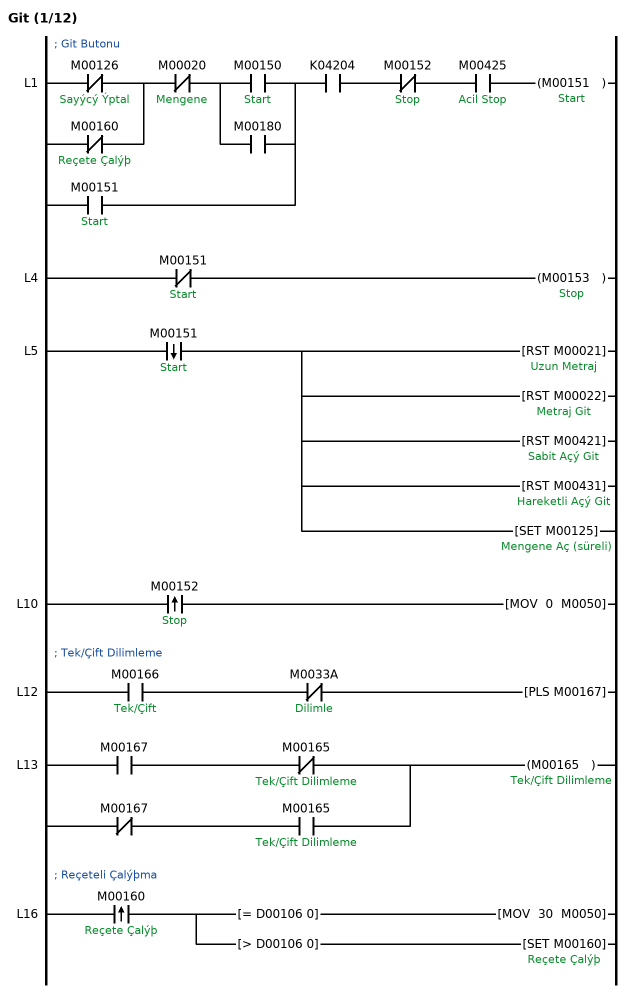
// Git Butonu
; L1
LOAD NOT  M00126	// Sayýcý Ýptal
OR NOT    M00160	// Reçete Çalýþ
AND NOT   M00020	// Mengene
LOAD      M00150	// Start
OR        M00180
AND LOAD
OR        M00151	// Start
AND       K04204
AND NOT   M00152	// Stop
AND       M00425	// Acil Stop
OUT       M00151	// Start
; L4
LOAD NOT  M00151	// Start
OUT       M00153	// Stop
; L5
LOADN     M00151	// Start
RST       M00021	// Uzun Metraj
RST       M00022	// Metraj Git
RST       M00421	// Sabit Açý Git
RST       M00431	// Hareketli Açý Git
SET       M00125	// Mengene Aç (süreli)
; L10
LOADP     M00152	// Stop
MOV       0 M0050
// Tek/Çift Dilimleme
; L12
LOAD      M00166	// Tek/Çift
AND NOT   M0033A	// Dilimle
OUTP      M00167
; L13
LOAD      M00167
AND NOT   M00165	// Tek/Çift Dilimleme
LOAD NOT  M00167
AND       M00165	// Tek/Çift Dilimleme
OR LOAD
OUT       M00165	// Tek/Çift Dilimleme
// Reçeteli Çalýþma
; L16
LOADP     M00160	// Reçete Çalýþ
MPUSH
AND=      D00106 0
MOV       30 M0050
MPOP
AND>      D00106 0
SET       M00160	// Reçete Çalýþ

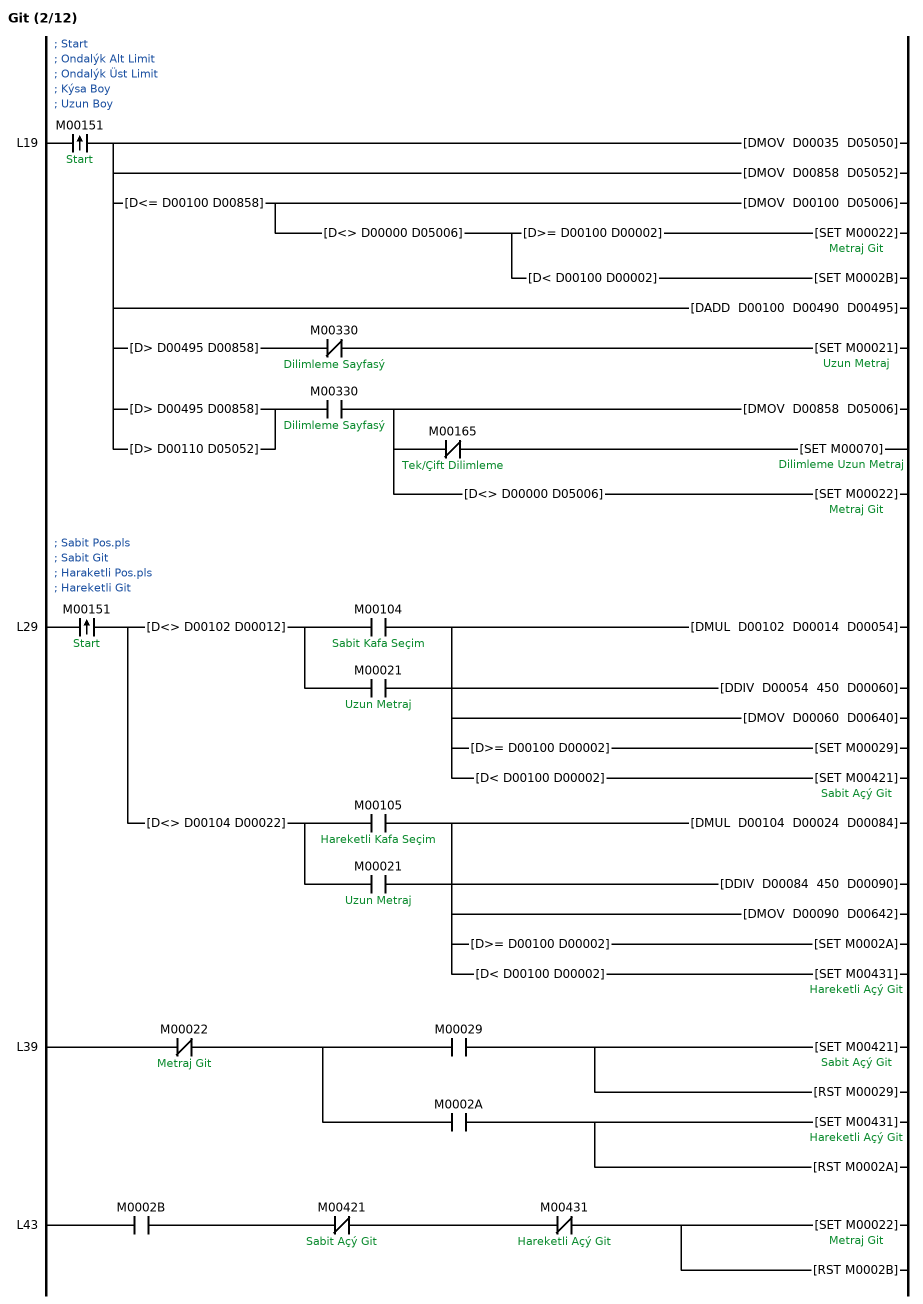
// Start
; L19
LOADP     M00151	// Start
DMOV      D00035 D05050
DMOV      D00858 D05052
MPUSH
ANDD<=    D00100 D00858
DMOV      D00100 D05006
ANDD<>    D00000 D05006
MPUSH
ANDD>=    D00100 D00002
SET       M00022	// Metraj Git
MPOP
ANDD<     D00100 D00002
SET       M0002B
MLOAD
DADD      D00100 D00490 D00495
ANDD>     D00495 D00858
AND NOT   M00330	// Dilimleme Sayfasý
SET       M00021	// Uzun Metraj
MPOP
LOADD>    D00495 D00858
ORD>      D00110 D05052
AND LOAD
AND       M00330	// Dilimleme Sayfasý
DMOV      D00858 D05006
MPUSH
AND NOT   M00165	// Tek/Çift Dilimleme
SET       M00070	// Dilimleme Uzun Metraj
MPOP
ANDD<>    D00000 D05006
SET       M00022	// Metraj Git
// output comment: Ondalýk Alt Limit
// output comment: Ondalýk Üst Limit
// output comment: Kýsa Boy
// output comment: Uzun Boy
; L29
LOADP     M00151	// Start
MPUSH
ANDD<>    D00102 D00012
LOAD      M00104	// Sabit Kafa Seçim
OR        M00021	// Uzun Metraj
AND LOAD
DMUL      D00102 D00014 D00054
DDIV      D00054 450 D00060
DMOV      D00060 D00640
MPUSH
ANDD>=    D00100 D00002
SET       M00029
MPOP
ANDD<     D00100 D00002
SET       M00421	// Sabit Açý Git
MPOP
ANDD<>    D00104 D00022
LOAD      M00105	// Hareketli Kafa Seçim
OR        M00021	// Uzun Metraj
AND LOAD
DMUL      D00104 D00024 D00084
DDIV      D00084 450 D00090
DMOV      D00090 D00642
MPUSH
ANDD>=    D00100 D00002
SET       M0002A
MPOP
ANDD<     D00100 D00002
SET       M00431	// Hareketli Açý Git
// output comment: Sabit Pos.pls
// output comment: Sabit Git
// output comment: Haraketli Pos.pls
// output comment: Hareketli Git
; L39
LOAD NOT  M00022	// Metraj Git
MPUSH
AND       M00029
SET       M00421	// Sabit Açý Git
RST       M00029
MPOP
AND       M0002A
SET       M00431	// Hareketli Açý Git
RST       M0002A
; L43
LOAD      M0002B
AND NOT   M00421	// Sabit Açý Git
AND NOT   M00431	// Hareketli Açý Git
SET       M00022	// Metraj Git
RST       M0002B

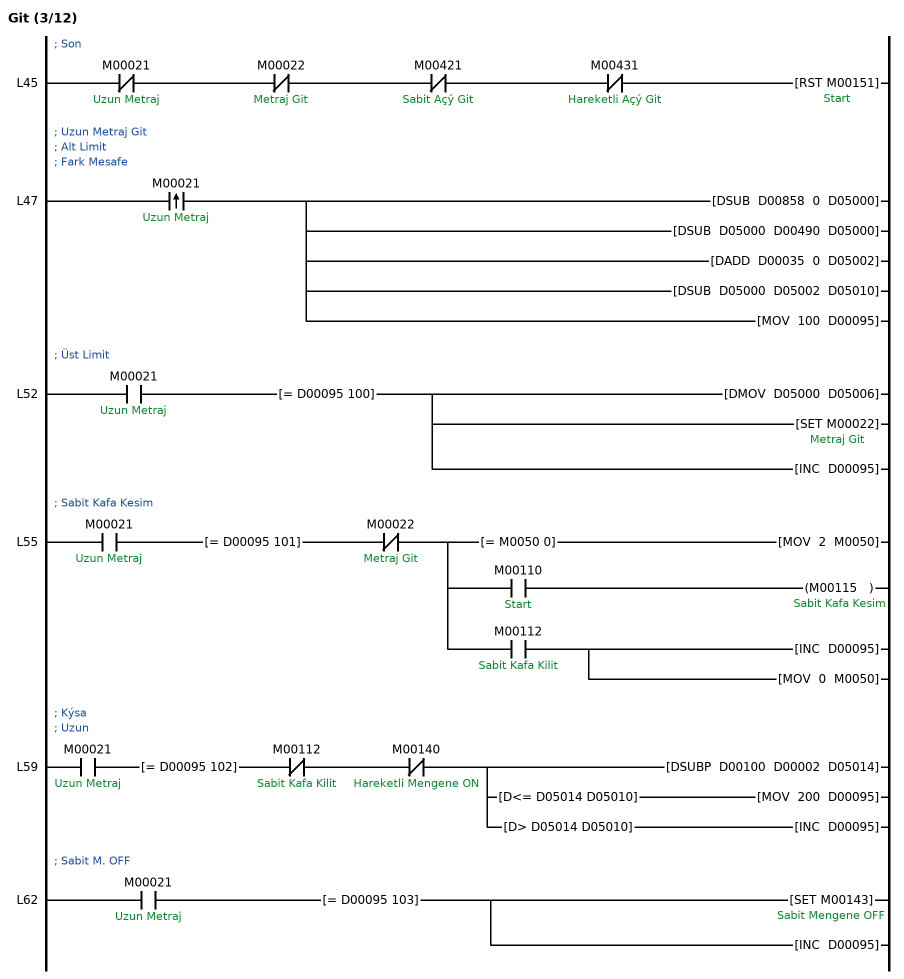
; L45
LOAD NOT  M00021	// Uzun Metraj
AND NOT   M00022	// Metraj Git
AND NOT   M00421	// Sabit Açý Git
AND NOT   M00431	// Hareketli Açý Git
RST       M00151	// Start
// output comment: Son
// Uzun Metraj Git
; L47
LOADP     M00021	// Uzun Metraj
DSUB      D00858 0 D05000
DSUB      D05000 D00490 D05000
DADD      D00035 0 D05002
DSUB      D05000 D05002 D05010
MOV       100 D00095
// output comment: Alt Limit
// output comment: Fark Mesafe
; L52
LOAD      M00021	// Uzun Metraj
AND=      D00095 100
DMOV      D05000 D05006
SET       M00022	// Metraj Git
INC       D00095
// output comment: Üst Limit
; L55
LOAD      M00021	// Uzun Metraj
AND=      D00095 101
AND NOT   M00022	// Metraj Git
MPUSH
AND=      M0050 0
MOV       2 M0050
MLOAD
AND       M00110	// Start
OUT       M00115	// Sabit Kafa Kesim
MPOP
AND       M00112	// Sabit Kafa Kilit
INC       D00095
MOV       0 M0050
// output comment: Sabit Kafa Kesim
; L59
LOAD      M00021	// Uzun Metraj
AND=      D00095 102
AND NOT   M00112	// Sabit Kafa Kilit
AND NOT   M00140	// Hareketli Mengene ON
DSUBP     D00100 D00002 D05014
MPUSH
ANDD<=    D05014 D05010
MOV       200 D00095
MPOP
ANDD>     D05014 D05010
INC       D00095
// output comment: Kýsa
// output comment: Uzun
; L62
LOAD      M00021	// Uzun Metraj
AND=      D00095 103
SET       M00143	// Sabit Mengene OFF
INC       D00095
// output comment: Sabit M. OFF

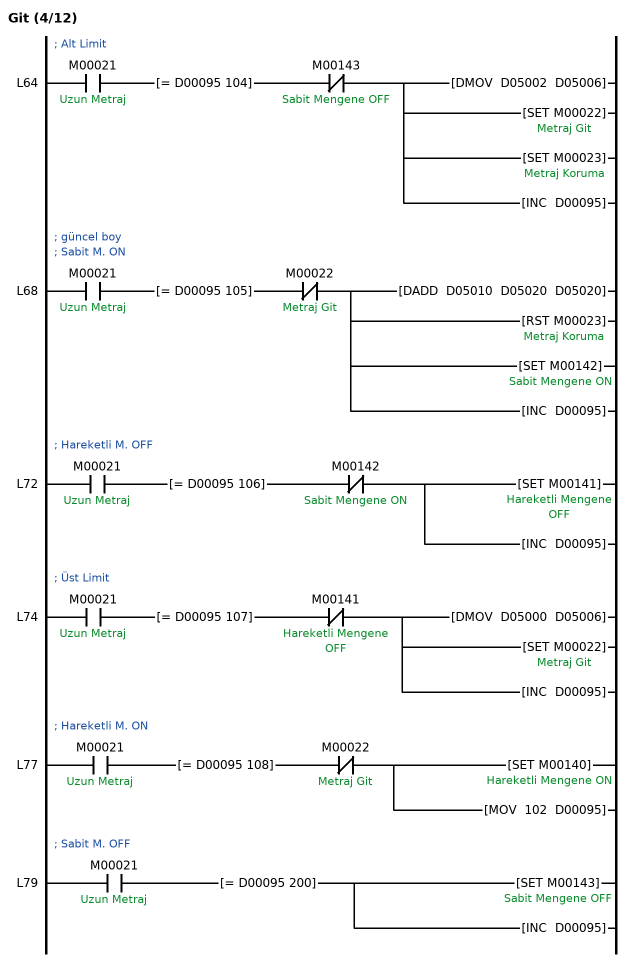
; L64
LOAD      M00021	// Uzun Metraj
AND=      D00095 104
AND NOT   M00143	// Sabit Mengene OFF
DMOV      D05002 D05006
SET       M00022	// Metraj Git
SET       M00023	// Metraj Koruma
INC       D00095
// output comment: Alt Limit
; L68
LOAD      M00021	// Uzun Metraj
AND=      D00095 105
AND NOT   M00022	// Metraj Git
DADD      D05010 D05020 D05020
RST       M00023	// Metraj Koruma
SET       M00142	// Sabit Mengene ON
INC       D00095
// output comment: güncel boy
// output comment: Sabit M. ON
; L72
LOAD      M00021	// Uzun Metraj
AND=      D00095 106
AND NOT   M00142	// Sabit Mengene ON
SET       M00141	// Hareketli Mengene OFF
INC       D00095
// output comment: Hareketli M. OFF
; L74
LOAD      M00021	// Uzun Metraj
AND=      D00095 107
AND NOT   M00141	// Hareketli Mengene OFF
DMOV      D05000 D05006
SET       M00022	// Metraj Git
INC       D00095
// output comment: Üst Limit
; L77
LOAD      M00021	// Uzun Metraj
AND=      D00095 108
AND NOT   M00022	// Metraj Git
SET       M00140	// Hareketli Mengene ON
MOV       102 D00095
// output comment: Hareketli M. ON
; L79
LOAD      M00021	// Uzun Metraj
AND=      D00095 200
SET       M00143	// Sabit Mengene OFF
INC       D00095
// output comment: Sabit M. OFF

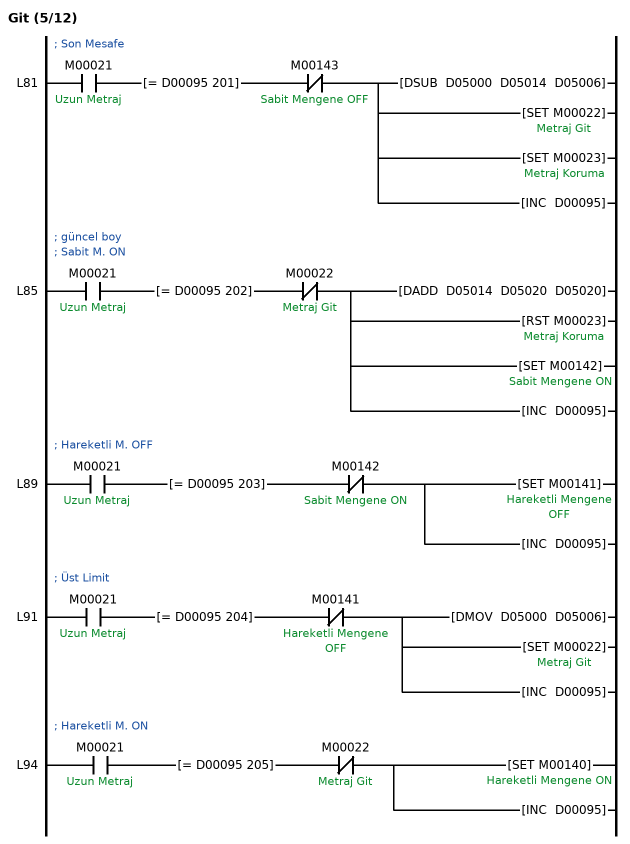
; L81
LOAD      M00021	// Uzun Metraj
AND=      D00095 201
AND NOT   M00143	// Sabit Mengene OFF
DSUB      D05000 D05014 D05006
SET       M00022	// Metraj Git
SET       M00023	// Metraj Koruma
INC       D00095
// output comment: Son Mesafe
; L85
LOAD      M00021	// Uzun Metraj
AND=      D00095 202
AND NOT   M00022	// Metraj Git
DADD      D05014 D05020 D05020
RST       M00023	// Metraj Koruma
SET       M00142	// Sabit Mengene ON
INC       D00095
// output comment: güncel boy
// output comment: Sabit M. ON
; L89
LOAD      M00021	// Uzun Metraj
AND=      D00095 203
AND NOT   M00142	// Sabit Mengene ON
SET       M00141	// Hareketli Mengene OFF
INC       D00095
// output comment: Hareketli M. OFF
; L91
LOAD      M00021	// Uzun Metraj
AND=      D00095 204
AND NOT   M00141	// Hareketli Mengene OFF
DMOV      D05000 D05006
SET       M00022	// Metraj Git
INC       D00095
// output comment: Üst Limit
; L94
LOAD      M00021	// Uzun Metraj
AND=      D00095 205
AND NOT   M00022	// Metraj Git
SET       M00140	// Hareketli Mengene ON
INC       D00095
// output comment: Hareketli M. ON

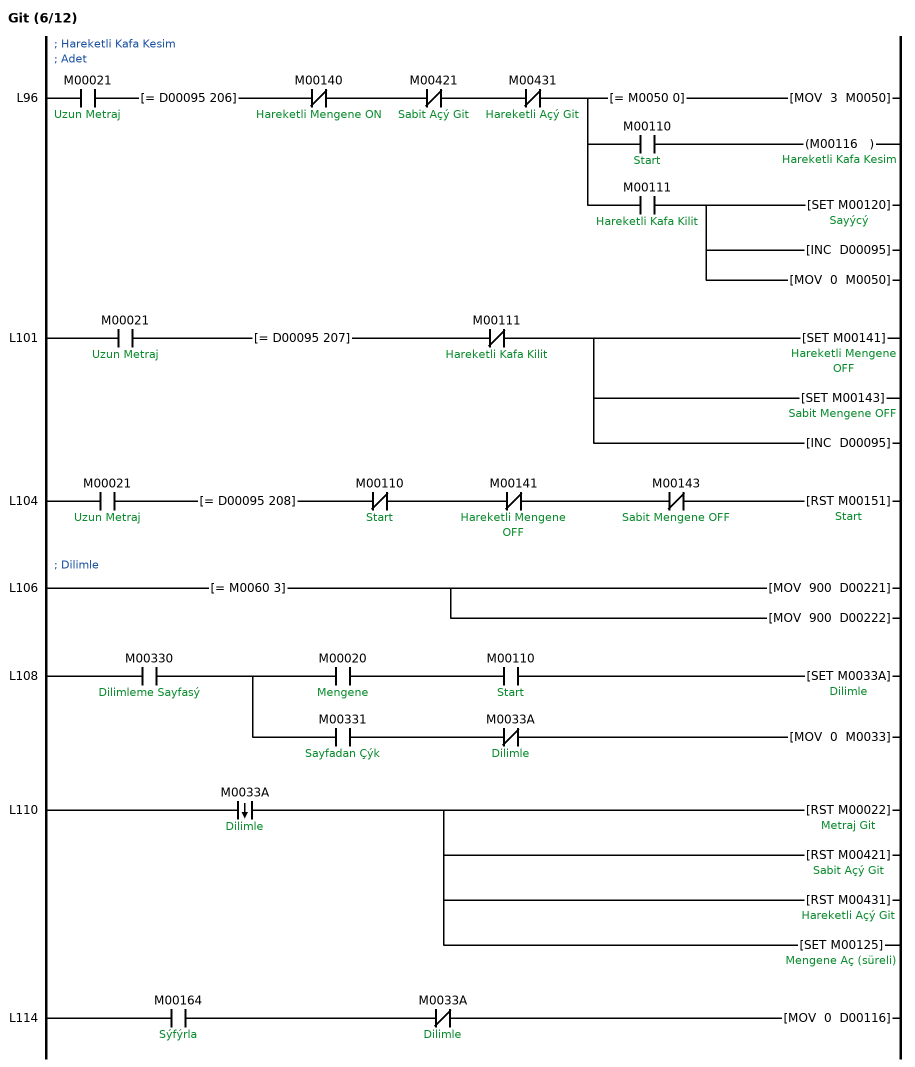
; L96
LOAD      M00021	// Uzun Metraj
AND=      D00095 206
AND NOT   M00140	// Hareketli Mengene ON
AND NOT   M00421	// Sabit Açý Git
AND NOT   M00431	// Hareketli Açý Git
MPUSH
AND=      M0050 0
MOV       3 M0050
MLOAD
AND       M00110	// Start
OUT       M00116	// Hareketli Kafa Kesim
MPOP
AND       M00111	// Hareketli Kafa Kilit
SET       M00120	// Sayýcý
INC       D00095
MOV       0 M0050
// output comment: Hareketli Kafa Kesim
// output comment: Adet
; L101
LOAD      M00021	// Uzun Metraj
AND=      D00095 207
AND NOT   M00111	// Hareketli Kafa Kilit
SET       M00141	// Hareketli Mengene OFF
SET       M00143	// Sabit Mengene OFF
INC       D00095
; L104
LOAD      M00021	// Uzun Metraj
AND=      D00095 208
AND NOT   M00110	// Start
AND NOT   M00141	// Hareketli Mengene OFF
AND NOT   M00143	// Sabit Mengene OFF
RST       M00151	// Start
// Dilimle
; L106
LOAD=     M0060 3
MOV       900 D00221
MOV       900 D00222
; L108
LOAD      M00330	// Dilimleme Sayfasý
MPUSH
AND       M00020	// Mengene
AND       M00110	// Start
SET       M0033A	// Dilimle
MPOP
AND       M00331	// Sayfadan Çýk
AND NOT   M0033A	// Dilimle
MOV       0 M0033
; L110
LOADN     M0033A	// Dilimle
RST       M00022	// Metraj Git
RST       M00421	// Sabit Açý Git
RST       M00431	// Hareketli Açý Git
SET       M00125	// Mengene Aç (süreli)
; L114
LOAD      M00164	// Sýfýrla
AND NOT   M0033A	// Dilimle
MOV       0 D00116

